# EPICS substitutions: iocBoot/iocvirPV/DPU09.substitutions
file "../../db/virAi.template"{ pattern
{DPU,    num,    Temp}
{09,    0,    500}
{09,    1,    500}
{09,    2,    500}
{09,    3,    500}
{09,    4,    500}
{09,    5,    500}
{09,    6,    500}
{09,    7,    500}
{09,    8,    500}
{09,    9,    500}
{09,    10,    500}
{09,    11,    500}
{09,    12,    500}
{09,    13,    500}
{09,    14,    500}
{09,    15,    500}
{09,    16,    500}
{09,    17,    500}
{09,    18,    500}
{09,    19,    500}
{09,    20,    500}
{09,    21,    500}
{09,    22,    500}
{09,    23,    500}
{09,    24,    500}
{09,    25,    500}
{09,    26,    500}
{09,    27,    500}
{09,    28,    500}
{09,    29,    500}
{09,    30,    500}
{09,    31,    500}
{09,    32,    500}
{09,    33,    500}
{09,    34,    500}
{09,    35,    500}
{09,    36,    500}
{09,    37,    500}
{09,    38,    500}
{09,    39,    500}
{09,    40,    500}
{09,    41,    500}
{09,    42,    500}
{09,    43,    500}
{09,    44,    500}
{09,    45,    500}
{09,    46,    500}
{09,    47,    500}
{09,    48,    500}
{09,    49,    500}
{09,    50,    500}
{09,    51,    500}
{09,    52,    500}
{09,    53,    500}
{09,    54,    500}
{09,    55,    500}
{09,    56,    500}
{09,    57,    500}
{09,    58,    500}
{09,    59,    500}
{09,    60,    500}
{09,    61,    500}
{09,    62,    500}
{09,    63,    500}
{09,    64,    500}
{09,    65,    500}
{09,    66,    500}
{09,    67,    500}
{09,    68,    500}
{09,    69,    500}
{09,    70,    500}
{09,    71,    500}
{09,    72,    500}
{09,    73,    500}
{09,    74,    500}
{09,    75,    500}
{09,    76,    500}
{09,    77,    500}
{09,    78,    500}
{09,    79,    500}
{09,    80,    500}
{09,    81,    500}
{09,    82,    500}
{09,    83,    500}
{09,    84,    500}
{09,    85,    500}
{09,    86,    500}
{09,    87,    500}
{09,    88,    500}
{09,    89,    500}
{09,    90,    500}
{09,    91,    500}
{09,    92,    500}
{09,    93,    500}
{09,    94,    500}
{09,    95,    500}
{09,    96,    500}
{09,    97,    500}
{09,    98,    500}
{09,    99,    500}
{09,    100,    500}
{09,    101,    500}
{09,    102,    500}
{09,    103,    500}
{09,    104,    500}
{09,    105,    500}
{09,    106,    500}
{09,    107,    500}
{09,    108,    500}
{09,    109,    500}
{09,    110,    500}
{09,    111,    500}
{09,    112,    500}
{09,    113,    500}
{09,    114,    500}
{09,    115,    500}
{09,    116,    500}
{09,    117,    500}
{09,    118,    500}
{09,    119,    500}
{09,    120,    500}
{09,    121,    500}
{09,    122,    500}
{09,    123,    500}
{09,    124,    500}
{09,    125,    500}
{09,    126,    500}
{09,    127,    500}
{09,    128,    500}
{09,    129,    500}
{09,    130,    500}
{09,    131,    500}
{09,    132,    500}
{09,    133,    500}
{09,    134,    500}
{09,    135,    500}
{09,    136,    500}
{09,    137,    500}
{09,    138,    500}
{09,    139,    500}
{09,    140,    500}
{09,    141,    500}
{09,    142,    500}
{09,    143,    500}
{09,    144,    500}
{09,    145,    500}
{09,    146,    500}
{09,    147,    500}
{09,    148,    500}
{09,    149,    500}
{09,    150,    500}
{09,    151,    500}
{09,    152,    500}
{09,    153,    500}
{09,    154,    500}
{09,    155,    500}
{09,    156,    500}
{09,    157,    500}
{09,    158,    500}
{09,    159,    500}
{09,    160,    500}
{09,    161,    500}
{09,    162,    500}
{09,    163,    500}
{09,    164,    500}
{09,    165,    500}
{09,    166,    500}
{09,    167,    500}
{09,    168,    500}
{09,    169,    500}
{09,    170,    500}
{09,    171,    500}
{09,    172,    500}
{09,    173,    500}
{09,    174,    500}
{09,    175,    500}
{09,    176,    500}
{09,    177,    500}
{09,    178,    500}
{09,    179,    500}
{09,    180,    500}
{09,    181,    500}
{09,    182,    500}
{09,    183,    500}
{09,    184,    500}
{09,    185,    500}
{09,    186,    500}
{09,    187,    500}
{09,    188,    500}
{09,    189,    500}
{09,    190,    500}
{09,    191,    500}
{09,    192,    500}
{09,    193,    500}
{09,    194,    500}
{09,    195,    500}
{09,    196,    500}
{09,    197,    500}
{09,    198,    500}
{09,    199,    500}
}
